// TIA Portal V20 export
TYPE "UDT_Service_ServReportParameter"
   STRUCT
      Analog : Array[0..31] of "UDT_MTP_AnaReportValue";
      Digital : Array[0..7] of "UDT_MTP_DIntReportValue";
      Binary : Array[0..31] of "UDT_MTP_BinReportValue";
      "String" : Array[0..7] of "UDT_MTP_StringReportValue";
   END_STRUCT;
END_TYPE
